// Mitsubishi GX Works2 project: BCD   PLC: Q03UDV

PROGRAM MAIN
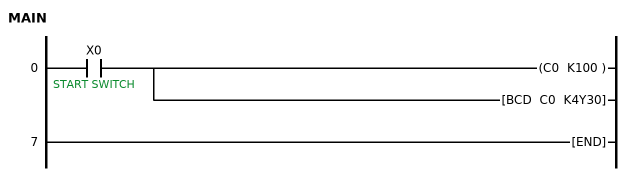
0     LD      X0  ; START SWITCH
      OUT     C0 K100
      BCD     C0 K4Y30
7     END
END_PROGRAM

// device comments not shown above
X1  ; DOOR OPEN SENSOR
Y20  ; ROBOTT START SIGNAL
Y21  ; OPERATION LAMP
Y22  ; STOP LAMP
